(* PLC project Adressering.ecp, WAGO e!COCKPIT e!COCKPIT *)
(* stored: creationDateTime 2021-01-18T14:20:23.2110188, modificationDateTime 2021-01-18T11:51:27.6823754 *)

TYPE typVAV : STRUCT
  xReady : BOOL;  (* Status adr. *)
  xEnable : BOOL;  (* Enable MP blokk *)
  xAddress : BOOL;  (* Adresserer VAV *)
  xFailed : BOOL;  (* Tilbakemelding adressering (True = SerieNr inn og ut ikke stemmer) *)
  sSetStatus : STRING;  (* Status tilbakemelding naar adresseringen er i SET step *)
  sGetStatus : STRING;  (* Status tilbakemelding naar adresseringen er i GET step *)
  iSerialNr : typSerialNo;  (* Serie NR *)
  bPort : BYTE;  (* VAV Port *)
  bAddress : BYTE;  (* VAV Address *)
  rAirVolume_SP : REAL;  (* Settpunkt 0-100% *)
  rOutPosition : REAL;  (* Vinkel *)
  rOutAirVolume_perc : REAL;  (* Luftmengde i prosent *)
  rOutAirVolume_m3h : REAL;  (* Luftmengde i m3h *)
  wSensorValue : WORD;
  rVmin : REAL;
  rVmax : REAL;  (* Max vinkel *)
  xControlRangeIncreased : BOOL;
  xMecanicalOverload : BOOL;
  xActuatorHunting : BOOL;
  xSensorError : BOOL;
  xManualOpen : BOOL;
  xManualClose : BOOL;
  vMin : REAL;  (* Min luftmengde SP / 0-100 *)
  vNorm : REAL;  (* Settpunkt ved bevegelse / 0-100 *)
  vMax : REAL;  (* Maks luftmengde SP / 0-100 *)
  vSize : REAL;  (* Max kubikk *)
  vSetpoint_m3h : REAL;  (* SP% *)
  xdontoptimize : BOOL;  (* Fjerner VAV fra Optimizer *)
END_STRUCT;
END_TYPE

{attribute 'qualified_only'}
VAR_GLOBAL  (* STLV59_360 *)
  STLV59_A_360_001_OU001_SQ401_Max : REAL;  (* Max spjeldvinkel tilluft *)
  STLV59_A_360_001_OU001_SQ501_Max : REAL;  (* max spjeldvinkel avtrekk *)
  STLV59_A_360_002_SQ401 : typVAV := (xEnable := TRUE, vMin := 125, vNorm := 250, vMax := 500, vSize := 1060, bPort := 1, bAddress := 1, iSerialNr := (wYearAndWeek := 0, wDayAndNumber := 0, bTypeID := 0, bTestStation := 0));  (* / *)
  STLV59_A_360_014_SQ401 : typVAV := (xEnable := TRUE, vMin := 75, vNorm := 0, vMax := 300, vSize := 434, bPort := 1, bAddress := 2, iSerialNr := (wYearAndWeek := 0, wDayAndNumber := 0, bTypeID := 0, bTestStation := 0));  (* / *)
  STLV59_A_360_014_SQ501 : typVAV := (xEnable := TRUE, vMin := 75, vNorm := 0, vMax := 300, vSize := 434, bPort := 1, bAddress := 3, iSerialNr := (wYearAndWeek := 0, wDayAndNumber := 0, bTypeID := 0, bTestStation := 0));  (* / *)
  STLV59_A_360_103_SQ401 : typVAV := (xEnable := TRUE, vMin := 375, vNorm := 0, vMax := 1500, vSize := 3619, bPort := 1, bAddress := 4, iSerialNr := (wYearAndWeek := 0, wDayAndNumber := 0, bTypeID := 0, bTestStation := 0));  (* / *)
  STLV59_A_360_103_SQ402 : typVAV := (xEnable := TRUE, vMin := 375, vNorm := 0, vMax := 1500, vSize := 3619, bPort := 1, bAddress := 5, iSerialNr := (wYearAndWeek := 0, wDayAndNumber := 0, bTypeID := 0, bTestStation := 0));  (* / *)
  STLV59_A_360_103_SQ501 : typVAV := (xEnable := TRUE, vMin := 375, vNorm := 0, vMax := 1500, vSize := 3619, bPort := 1, bAddress := 6, iSerialNr := (wYearAndWeek := 0, wDayAndNumber := 0, bTypeID := 0, bTestStation := 0));  (* / *)
  STLV59_A_360_103_SQ502 : typVAV := (xEnable := TRUE, vMin := 375, vNorm := 0, vMax := 1500, vSize := 3619, bPort := 1, bAddress := 7, iSerialNr := (wYearAndWeek := 0, wDayAndNumber := 0, bTypeID := 0, bTestStation := 0));  (* / *)
  STLV59_A_360_002_SQ402 : typVAV := (xEnable := TRUE, vMin := 175, vNorm := 0, vMax := 700, vSize := 1060, bPort := 2, bAddress := 1, iSerialNr := (wYearAndWeek := 0, wDayAndNumber := 0, bTypeID := 0, bTestStation := 0));  (* / *)
  STLV59_A_360_002_SQ501 : typVAV := (xEnable := TRUE, vMin := 125, vNorm := 250, vMax := 500, vSize := 1060, bPort := 2, bAddress := 2, iSerialNr := (wYearAndWeek := 0, wDayAndNumber := 0, bTypeID := 0, bTestStation := 0));  (* / *)
  STLV59_A_360_002_SQ502 : typVAV := (xEnable := TRUE, vMin := 175, vNorm := 0, vMax := 700, vSize := 1060, bPort := 2, bAddress := 3, iSerialNr := (wYearAndWeek := 0, wDayAndNumber := 0, bTypeID := 0, bTestStation := 0));  (* / *)
  STLV59_A_360_006_SQ401 : typVAV := (xEnable := TRUE, vMin := 188, vNorm := 0, vMax := 750, vSize := 1060, bPort := 2, bAddress := 4, iSerialNr := (wYearAndWeek := 0, wDayAndNumber := 0, bTypeID := 0, bTestStation := 0));  (* / *)
  STLV59_A_360_008_SQ501 : typVAV := (xEnable := TRUE, vMin := 188, vNorm := 0, vMax := 750, vSize := 1060, bPort := 2, bAddress := 5, iSerialNr := (wYearAndWeek := 0, wDayAndNumber := 0, bTypeID := 0, bTestStation := 0));  (* / *)
  STLV59_A_360_011_SQ401 : typVAV := (xEnable := TRUE, vMin := 50, vNorm := 0, vMax := 200, vSize := 700, bPort := 2, bAddress := 6, iSerialNr := (wYearAndWeek := 0, wDayAndNumber := 0, bTypeID := 0, bTestStation := 0));  (* / *)
  STLV59_A_360_011_SQ501 : typVAV := (xEnable := TRUE, vMin := 50, vNorm := 0, vMax := 200, vSize := 265, bPort := 2, bAddress := 7, iSerialNr := (wYearAndWeek := 0, wDayAndNumber := 0, bTypeID := 0, bTestStation := 0));  (* / *)
  STLV59_A_360_T1U_SQ401 : typVAV := (xEnable := TRUE, vMin := 50, vNorm := 0, vMax := 200, vSize := 434, bPort := 2, bAddress := 8, iSerialNr := (wYearAndWeek := 0, wDayAndNumber := 0, bTypeID := 0, bTestStation := 0));  (* / *)
  STLV59_A_360_001_SQ401 : typVAV := (xEnable := TRUE, vMin := 25, vNorm := 100, vMax := 100, vSize := 265, bPort := 3, bAddress := 1, iSerialNr := (wYearAndWeek := 0, wDayAndNumber := 0, bTypeID := 0, bTestStation := 0));  (* / *)
  STLV59_A_360_001_SQ501 : typVAV := (xEnable := TRUE, vMin := 25, vNorm := 100, vMax := 100, vSize := 265, bPort := 3, bAddress := 2, iSerialNr := (wYearAndWeek := 0, wDayAndNumber := 0, bTypeID := 0, bTestStation := 0));  (* / *)
  STLV59_A_360_109_SQ401 : typVAV := (xEnable := TRUE, vMin := 200, vNorm := 200, vMax := 200, vSize := 434, bPort := 3, bAddress := 3, iSerialNr := (wYearAndWeek := 0, wDayAndNumber := 0, bTypeID := 0, bTestStation := 0));  (* / *)
  STLV59_A_360_110_SQ501 : typVAV := (xEnable := TRUE, vMin := 200, vNorm := 200, vMax := 200, vSize := 265, bPort := 3, bAddress := 4, iSerialNr := (wYearAndWeek := 0, wDayAndNumber := 0, bTypeID := 0, bTestStation := 0));  (* / *)
  STLV59_A_360_212_SQ401 : typVAV := (xEnable := TRUE, vMin := 63, vNorm := 0, vMax := 250, vSize := 700, bPort := 3, bAddress := 5, iSerialNr := (wYearAndWeek := 0, wDayAndNumber := 0, bTypeID := 0, bTestStation := 0));  (* / *)
  STLV59_A_360_212_SQ501 : typVAV := (xEnable := TRUE, vMin := 63, vNorm := 0, vMax := 250, vSize := 700, bPort := 3, bAddress := 6, iSerialNr := (wYearAndWeek := 0, wDayAndNumber := 0, bTypeID := 0, bTestStation := 0));  (* / *)
  STLV59_A_360_213_SQ401 : typVAV := (xEnable := TRUE, vMin := 138, vNorm := 0, vMax := 550, vSize := 70, bPort := 3, bAddress := 7, iSerialNr := (wYearAndWeek := 0, wDayAndNumber := 0, bTypeID := 0, bTestStation := 0));  (* / *)
  STLV59_A_360_213_SQ501 : typVAV := (xEnable := TRUE, vMin := 138, vNorm := 0, vMax := 550, vSize := 265, bPort := 3, bAddress := 8, iSerialNr := (wYearAndWeek := 0, wDayAndNumber := 0, bTypeID := 0, bTestStation := 0));  (* / *)
END_VAR

FUNCTION_BLOCK fbAutAd
  VAR_INPUT
    iSerialNr : typSerialNo;
    bPort : BYTE;
    bAddress : BYTE;
    xReset : BOOL;
    xNext : BOOL;
  END_VAR
  VAR_OUTPUT
    i : INT := 0;
    xFailed : BOOL;
    sSetStatus : STRING;
    sGetStatus : STRING;
  END_VAR
  VAR
    xLearn : BOOL;
    xRetry : BOOL;
    VAV_Addressing : fbMpBusAddressing;
  END_VAR

	//Resetter forgje VAVs verdier
	IF xReset THEN
		i:= 0;
		xRetry:= FALSE;
		xFailed:= FALSE;
		sSetStatus:= '';
		sGetStatus:= '';

//Begynner paa neste VAV
	ELSIF i<1 AND xNext THEN
		VAV_Addressing
		(
			bPortMpBus:= bPort,
			bAddress:= bAddress,
			typINSerialNo:= iSerialNr,
			xLearn:= xLearn
		);
		i:= 1;

//Skriver rett port og adresse til VAV naar blokken er klar
	ELSIF VAV_Addressing.xReady AND i=1 THEN
		VAV_Addressing
		(
			xSet:= TRUE,
			xLearn:= xLearn
		);
		i:= 2;

//Spoer etter serie nr som hoerer til port og adresse
	ELSIF VAV_Addressing.xReady AND i=2 THEN
		sSetStatus:= VAV_Addressing.sStatus;
		VAV_Addressing
		(
			xGetSerialNO:= TRUE,
			xLearn:= xLearn
		);
		i:= 3;

//Sjekker om serie nr. som tilhoerer port og adressen stemmer
	ELSIF VAV_Addressing.xReady AND i=3 THEN
		sGetStatus:= VAV_Addressing.sStatus;
		//Sjekker om serie nr stemmer
		IF xRetry AND VAV_Addressing.typOUTSerialNo.wYearAndWeek <> iSerialNr.wYearAndWeek OR VAV_Addressing.typOUTSerialNo.wDayAndNumber <> iSerialNr.wDayAndNumber OR VAV_Addressing.typOUTSerialNo.bTypeID <> iSerialNr.bTypeID OR VAV_Addressing.typOUTSerialNo.bTestStation <> iSerialNr.bTestStation THEN
			xRetry:= FALSE;
			xFailed:= TRUE;
			i:=4;
		ELSIF VAV_Addressing.typOUTSerialNo.wYearAndWeek <> iSerialNr.wYearAndWeek OR VAV_Addressing.typOUTSerialNo.wDayAndNumber <> iSerialNr.wDayAndNumber OR VAV_Addressing.typOUTSerialNo.bTypeID <> iSerialNr.bTypeID OR VAV_Addressing.typOUTSerialNo.bTestStation <> iSerialNr.bTestStation THEN
			xRetry:= TRUE;
			i:=1;
		ELSE
			i:=4;
		END_IF

//Resetter xSet og xGet, og Setter Port, adresse og serie nr. og henter status
	ELSE
		VAV_Addressing
		(
			bPortMpBus:= bPort,
			bAddress:= bAddress,
			typINSerialNo:= iSerialNr,
			xLearn:= xLearn,
			xSet:= FALSE,
			xGetSerialNO:= FALSE,
			xLearn:= xLearn
		);
	END_IF
				
END_FUNCTION_BLOCK

PROGRAM PRG_360_VAV_Adressering
  VAR
    xReset : BOOL;
    xRun : BOOL;
    xInit : BOOL := TRUE;
    Auto : fbAutAd;
    iLinje : INT;  (* Linje som skal adresseres *)
    iVAV : INT := 1;  (* VAV(adr.) som adresseres *)
  END_VAR

					IF xReset THEN
	Auto(xReset:= TRUE);
	xInit:= TRUE;
	xReset:= FALSE;
ELSIF xRun THEN

	IF STLV59_360.STLV59_A_360_002_SQ401.xAddress OR (iLinje = 1 AND iVAV = 1) THEN

		IF xInit THEN
			STLV59_360.STLV59_A_360_002_SQ401.xEnable:= FALSE;
			Auto(
				bPort:= STLV59_360.STLV59_A_360_002_SQ401.bPort,
				bAddress:= STLV59_360.STLV59_A_360_002_SQ401.bAddress,
				iSerialNr:= STLV59_360.STLV59_A_360_002_SQ401.iSerialNr,
				xNext:= TRUE,
				xReset:= FALSE
				);
			xInit:= FALSE;

		ELSIF Auto.i=4 THEN
			STLV59_360.STLV59_A_360_002_SQ401.sSetStatus:= Auto.sSetStatus;
				STLV59_360.STLV59_A_360_002_SQ401.sGetStatus:= Auto.sGetStatus;
				STLV59_360.STLV59_A_360_002_SQ401.xFailed:= Auto.xFailed;
				STLV59_360.STLV59_A_360_002_SQ401.xAddress:= FALSE;
				STLV59_360.STLV59_A_360_002_SQ401.xEnable:= TRUE;
				xReset:= TRUE;
				iVAV:=iVAV+1;

			ELSE
				Auto(xNext:= FALSE);
			END_IF

	ELSIF STLV59_360.STLV59_A_360_014_SQ401.xAddress OR (iLinje = 1 AND iVAV = 2) THEN

		IF xInit THEN
			STLV59_360.STLV59_A_360_014_SQ401.xEnable:= FALSE;
			Auto(
				bPort:= STLV59_360.STLV59_A_360_014_SQ401.bPort,
				bAddress:= STLV59_360.STLV59_A_360_014_SQ401.bAddress,
				iSerialNr:= STLV59_360.STLV59_A_360_014_SQ401.iSerialNr,
				xNext:= TRUE,
				xReset:= FALSE
				);
			xInit:= FALSE;

		ELSIF Auto.i=4 THEN
			STLV59_360.STLV59_A_360_014_SQ401.sSetStatus:= Auto.sSetStatus;
				STLV59_360.STLV59_A_360_014_SQ401.sGetStatus:= Auto.sGetStatus;
				STLV59_360.STLV59_A_360_014_SQ401.xFailed:= Auto.xFailed;
				STLV59_360.STLV59_A_360_014_SQ401.xAddress:= FALSE;
				STLV59_360.STLV59_A_360_014_SQ401.xEnable:= TRUE;
				xReset:= TRUE;
				iVAV:=iVAV+1;

			ELSE
				Auto(xNext:= FALSE);
			END_IF

	ELSIF STLV59_360.STLV59_A_360_014_SQ501.xAddress OR (iLinje = 1 AND iVAV = 3) THEN

		IF xInit THEN
			STLV59_360.STLV59_A_360_014_SQ501.xEnable:= FALSE;
			Auto(
				bPort:= STLV59_360.STLV59_A_360_014_SQ501.bPort,
				bAddress:= STLV59_360.STLV59_A_360_014_SQ501.bAddress,
				iSerialNr:= STLV59_360.STLV59_A_360_014_SQ501.iSerialNr,
				xNext:= TRUE,
				xReset:= FALSE
				);
			xInit:= FALSE;

		ELSIF Auto.i=4 THEN
			STLV59_360.STLV59_A_360_014_SQ501.sSetStatus:= Auto.sSetStatus;
				STLV59_360.STLV59_A_360_014_SQ501.sGetStatus:= Auto.sGetStatus;
				STLV59_360.STLV59_A_360_014_SQ501.xFailed:= Auto.xFailed;
				STLV59_360.STLV59_A_360_014_SQ501.xAddress:= FALSE;
				STLV59_360.STLV59_A_360_014_SQ501.xEnable:= TRUE;
				xReset:= TRUE;
				iVAV:=iVAV+1;

			ELSE
				Auto(xNext:= FALSE);
			END_IF

	ELSIF STLV59_360.STLV59_A_360_103_SQ401.xAddress OR (iLinje = 1 AND iVAV = 4) THEN

		IF xInit THEN
			STLV59_360.STLV59_A_360_103_SQ401.xEnable:= FALSE;
			Auto(
				bPort:= STLV59_360.STLV59_A_360_103_SQ401.bPort,
				bAddress:= STLV59_360.STLV59_A_360_103_SQ401.bAddress,
				iSerialNr:= STLV59_360.STLV59_A_360_103_SQ401.iSerialNr,
				xNext:= TRUE,
				xReset:= FALSE
				);
			xInit:= FALSE;

		ELSIF Auto.i=4 THEN
			STLV59_360.STLV59_A_360_103_SQ401.sSetStatus:= Auto.sSetStatus;
				STLV59_360.STLV59_A_360_103_SQ401.sGetStatus:= Auto.sGetStatus;
				STLV59_360.STLV59_A_360_103_SQ401.xFailed:= Auto.xFailed;
				STLV59_360.STLV59_A_360_103_SQ401.xAddress:= FALSE;
				STLV59_360.STLV59_A_360_103_SQ401.xEnable:= TRUE;
				xReset:= TRUE;
				iVAV:=iVAV+1;

			ELSE
				Auto(xNext:= FALSE);
			END_IF

	ELSIF STLV59_360.STLV59_A_360_103_SQ402.xAddress OR (iLinje = 1 AND iVAV = 5) THEN

		IF xInit THEN
			STLV59_360.STLV59_A_360_103_SQ402.xEnable:= FALSE;
			Auto(
				bPort:= STLV59_360.STLV59_A_360_103_SQ402.bPort,
				bAddress:= STLV59_360.STLV59_A_360_103_SQ402.bAddress,
				iSerialNr:= STLV59_360.STLV59_A_360_103_SQ402.iSerialNr,
				xNext:= TRUE,
				xReset:= FALSE
				);
			xInit:= FALSE;

		ELSIF Auto.i=4 THEN
			STLV59_360.STLV59_A_360_103_SQ402.sSetStatus:= Auto.sSetStatus;
				STLV59_360.STLV59_A_360_103_SQ402.sGetStatus:= Auto.sGetStatus;
				STLV59_360.STLV59_A_360_103_SQ402.xFailed:= Auto.xFailed;
				STLV59_360.STLV59_A_360_103_SQ402.xAddress:= FALSE;
				STLV59_360.STLV59_A_360_103_SQ402.xEnable:= TRUE;
				xReset:= TRUE;
				iVAV:=iVAV+1;

			ELSE
				Auto(xNext:= FALSE);
			END_IF

	ELSIF STLV59_360.STLV59_A_360_103_SQ501.xAddress OR (iLinje = 1 AND iVAV = 6) THEN

		IF xInit THEN
			STLV59_360.STLV59_A_360_103_SQ501.xEnable:= FALSE;
			Auto(
				bPort:= STLV59_360.STLV59_A_360_103_SQ501.bPort,
				bAddress:= STLV59_360.STLV59_A_360_103_SQ501.bAddress,
				iSerialNr:= STLV59_360.STLV59_A_360_103_SQ501.iSerialNr,
				xNext:= TRUE,
				xReset:= FALSE
				);
			xInit:= FALSE;

		ELSIF Auto.i=4 THEN
			STLV59_360.STLV59_A_360_103_SQ501.sSetStatus:= Auto.sSetStatus;
				STLV59_360.STLV59_A_360_103_SQ501.sGetStatus:= Auto.sGetStatus;
				STLV59_360.STLV59_A_360_103_SQ501.xFailed:= Auto.xFailed;
				STLV59_360.STLV59_A_360_103_SQ501.xAddress:= FALSE;
				STLV59_360.STLV59_A_360_103_SQ501.xEnable:= TRUE;
				xReset:= TRUE;
				iVAV:=iVAV+1;

			ELSE
				Auto(xNext:= FALSE);
			END_IF

	ELSIF STLV59_360.STLV59_A_360_103_SQ502.xAddress OR (iLinje = 1 AND iVAV = 7) THEN

		IF xInit THEN
			STLV59_360.STLV59_A_360_103_SQ502.xEnable:= FALSE;
			Auto(
				bPort:= STLV59_360.STLV59_A_360_103_SQ502.bPort,
				bAddress:= STLV59_360.STLV59_A_360_103_SQ502.bAddress,
				iSerialNr:= STLV59_360.STLV59_A_360_103_SQ502.iSerialNr,
				xNext:= TRUE,
				xReset:= FALSE
				);
			xInit:= FALSE;

		ELSIF Auto.i=4 THEN
			STLV59_360.STLV59_A_360_103_SQ502.sSetStatus:= Auto.sSetStatus;
				STLV59_360.STLV59_A_360_103_SQ502.sGetStatus:= Auto.sGetStatus;
				STLV59_360.STLV59_A_360_103_SQ502.xFailed:= Auto.xFailed;
				STLV59_360.STLV59_A_360_103_SQ502.xAddress:= FALSE;
				STLV59_360.STLV59_A_360_103_SQ502.xEnable:= TRUE;
				xReset:= TRUE;
				iVAV:=iVAV+1;

			ELSE
				Auto(xNext:= FALSE);
			END_IF

	ELSIF STLV59_360.STLV59_A_360_002_SQ402.xAddress OR (iLinje = 2 AND iVAV = 1) THEN

		IF xInit THEN
			STLV59_360.STLV59_A_360_002_SQ402.xEnable:= FALSE;
			Auto(
				bPort:= STLV59_360.STLV59_A_360_002_SQ402.bPort,
				bAddress:= STLV59_360.STLV59_A_360_002_SQ402.bAddress,
				iSerialNr:= STLV59_360.STLV59_A_360_002_SQ402.iSerialNr,
				xNext:= TRUE,
				xReset:= FALSE
				);
			xInit:= FALSE;

		ELSIF Auto.i=4 THEN
			STLV59_360.STLV59_A_360_002_SQ402.sSetStatus:= Auto.sSetStatus;
				STLV59_360.STLV59_A_360_002_SQ402.sGetStatus:= Auto.sGetStatus;
				STLV59_360.STLV59_A_360_002_SQ402.xFailed:= Auto.xFailed;
				STLV59_360.STLV59_A_360_002_SQ402.xAddress:= FALSE;
				STLV59_360.STLV59_A_360_002_SQ402.xEnable:= TRUE;
				xReset:= TRUE;
				iVAV:=iVAV+1;

			ELSE
				Auto(xNext:= FALSE);
			END_IF

	ELSIF STLV59_360.STLV59_A_360_002_SQ501.xAddress OR (iLinje = 2 AND iVAV = 2) THEN

		IF xInit THEN
			STLV59_360.STLV59_A_360_002_SQ501.xEnable:= FALSE;
			Auto(
				bPort:= STLV59_360.STLV59_A_360_002_SQ501.bPort,
				bAddress:= STLV59_360.STLV59_A_360_002_SQ501.bAddress,
				iSerialNr:= STLV59_360.STLV59_A_360_002_SQ501.iSerialNr,
				xNext:= TRUE,
				xReset:= FALSE
				);
			xInit:= FALSE;

		ELSIF Auto.i=4 THEN
			STLV59_360.STLV59_A_360_002_SQ501.sSetStatus:= Auto.sSetStatus;
				STLV59_360.STLV59_A_360_002_SQ501.sGetStatus:= Auto.sGetStatus;
				STLV59_360.STLV59_A_360_002_SQ501.xFailed:= Auto.xFailed;
				STLV59_360.STLV59_A_360_002_SQ501.xAddress:= FALSE;
				STLV59_360.STLV59_A_360_002_SQ501.xEnable:= TRUE;
				xReset:= TRUE;
				iVAV:=iVAV+1;

			ELSE
				Auto(xNext:= FALSE);
			END_IF

	ELSIF STLV59_360.STLV59_A_360_002_SQ502.xAddress OR (iLinje = 2 AND iVAV = 3) THEN

		IF xInit THEN
			STLV59_360.STLV59_A_360_002_SQ502.xEnable:= FALSE;
			Auto(
				bPort:= STLV59_360.STLV59_A_360_002_SQ502.bPort,
				bAddress:= STLV59_360.STLV59_A_360_002_SQ502.bAddress,
				iSerialNr:= STLV59_360.STLV59_A_360_002_SQ502.iSerialNr,
				xNext:= TRUE,
				xReset:= FALSE
				);
			xInit:= FALSE;

		ELSIF Auto.i=4 THEN
			STLV59_360.STLV59_A_360_002_SQ502.sSetStatus:= Auto.sSetStatus;
				STLV59_360.STLV59_A_360_002_SQ502.sGetStatus:= Auto.sGetStatus;
				STLV59_360.STLV59_A_360_002_SQ502.xFailed:= Auto.xFailed;
				STLV59_360.STLV59_A_360_002_SQ502.xAddress:= FALSE;
				STLV59_360.STLV59_A_360_002_SQ502.xEnable:= TRUE;
				xReset:= TRUE;
				iVAV:=iVAV+1;

			ELSE
				Auto(xNext:= FALSE);
			END_IF

	ELSIF STLV59_360.STLV59_A_360_006_SQ401.xAddress OR (iLinje = 2 AND iVAV = 4) THEN

		IF xInit THEN
			STLV59_360.STLV59_A_360_006_SQ401.xEnable:= FALSE;
			Auto(
				bPort:= STLV59_360.STLV59_A_360_006_SQ401.bPort,
				bAddress:= STLV59_360.STLV59_A_360_006_SQ401.bAddress,
				iSerialNr:= STLV59_360.STLV59_A_360_006_SQ401.iSerialNr,
				xNext:= TRUE,
				xReset:= FALSE
				);
			xInit:= FALSE;

		ELSIF Auto.i=4 THEN
			STLV59_360.STLV59_A_360_006_SQ401.sSetStatus:= Auto.sSetStatus;
				STLV59_360.STLV59_A_360_006_SQ401.sGetStatus:= Auto.sGetStatus;
				STLV59_360.STLV59_A_360_006_SQ401.xFailed:= Auto.xFailed;
				STLV59_360.STLV59_A_360_006_SQ401.xAddress:= FALSE;
				STLV59_360.STLV59_A_360_006_SQ401.xEnable:= TRUE;
				xReset:= TRUE;
				iVAV:=iVAV+1;

			ELSE
				Auto(xNext:= FALSE);
			END_IF

	ELSIF STLV59_360.STLV59_A_360_008_SQ501.xAddress OR (iLinje = 2 AND iVAV = 5) THEN

		IF xInit THEN
			STLV59_360.STLV59_A_360_008_SQ501.xEnable:= FALSE;
			Auto(
				bPort:= STLV59_360.STLV59_A_360_008_SQ501.bPort,
				bAddress:= STLV59_360.STLV59_A_360_008_SQ501.bAddress,
				iSerialNr:= STLV59_360.STLV59_A_360_008_SQ501.iSerialNr,
				xNext:= TRUE,
				xReset:= FALSE
				);
			xInit:= FALSE;

		ELSIF Auto.i=4 THEN
			STLV59_360.STLV59_A_360_008_SQ501.sSetStatus:= Auto.sSetStatus;
				STLV59_360.STLV59_A_360_008_SQ501.sGetStatus:= Auto.sGetStatus;
				STLV59_360.STLV59_A_360_008_SQ501.xFailed:= Auto.xFailed;
				STLV59_360.STLV59_A_360_008_SQ501.xAddress:= FALSE;
				STLV59_360.STLV59_A_360_008_SQ501.xEnable:= TRUE;
				xReset:= TRUE;
				iVAV:=iVAV+1;

			ELSE
				Auto(xNext:= FALSE);
			END_IF

	ELSIF STLV59_360.STLV59_A_360_011_SQ401.xAddress OR (iLinje = 2 AND iVAV = 6) THEN

		IF xInit THEN
			STLV59_360.STLV59_A_360_011_SQ401.xEnable:= FALSE;
			Auto(
				bPort:= STLV59_360.STLV59_A_360_011_SQ401.bPort,
				bAddress:= STLV59_360.STLV59_A_360_011_SQ401.bAddress,
				iSerialNr:= STLV59_360.STLV59_A_360_011_SQ401.iSerialNr,
				xNext:= TRUE,
				xReset:= FALSE
				);
			xInit:= FALSE;

		ELSIF Auto.i=4 THEN
			STLV59_360.STLV59_A_360_011_SQ401.sSetStatus:= Auto.sSetStatus;
				STLV59_360.STLV59_A_360_011_SQ401.sGetStatus:= Auto.sGetStatus;
				STLV59_360.STLV59_A_360_011_SQ401.xFailed:= Auto.xFailed;
				STLV59_360.STLV59_A_360_011_SQ401.xAddress:= FALSE;
				STLV59_360.STLV59_A_360_011_SQ401.xEnable:= TRUE;
				xReset:= TRUE;
				iVAV:=iVAV+1;

			ELSE
				Auto(xNext:= FALSE);
			END_IF

	ELSIF STLV59_360.STLV59_A_360_011_SQ501.xAddress OR (iLinje = 2 AND iVAV = 7) THEN

		IF xInit THEN
			STLV59_360.STLV59_A_360_011_SQ501.xEnable:= FALSE;
			Auto(
				bPort:= STLV59_360.STLV59_A_360_011_SQ501.bPort,
				bAddress:= STLV59_360.STLV59_A_360_011_SQ501.bAddress,
				iSerialNr:= STLV59_360.STLV59_A_360_011_SQ501.iSerialNr,
				xNext:= TRUE,
				xReset:= FALSE
				);
			xInit:= FALSE;

		ELSIF Auto.i=4 THEN
			STLV59_360.STLV59_A_360_011_SQ501.sSetStatus:= Auto.sSetStatus;
				STLV59_360.STLV59_A_360_011_SQ501.sGetStatus:= Auto.sGetStatus;
				STLV59_360.STLV59_A_360_011_SQ501.xFailed:= Auto.xFailed;
				STLV59_360.STLV59_A_360_011_SQ501.xAddress:= FALSE;
				STLV59_360.STLV59_A_360_011_SQ501.xEnable:= TRUE;
				xReset:= TRUE;
				iVAV:=iVAV+1;

			ELSE
				Auto(xNext:= FALSE);
			END_IF

	ELSIF STLV59_360.STLV59_A_360_T1U_SQ401.xAddress OR (iLinje = 2 AND iVAV = 8) THEN

		IF xInit THEN
			STLV59_360.STLV59_A_360_T1U_SQ401.xEnable:= FALSE;
			Auto(
				bPort:= STLV59_360.STLV59_A_360_T1U_SQ401.bPort,
				bAddress:= STLV59_360.STLV59_A_360_T1U_SQ401.bAddress,
				iSerialNr:= STLV59_360.STLV59_A_360_T1U_SQ401.iSerialNr,
				xNext:= TRUE,
				xReset:= FALSE
				);
			xInit:= FALSE;

		ELSIF Auto.i=4 THEN
			STLV59_360.STLV59_A_360_T1U_SQ401.sSetStatus:= Auto.sSetStatus;
				STLV59_360.STLV59_A_360_T1U_SQ401.sGetStatus:= Auto.sGetStatus;
				STLV59_360.STLV59_A_360_T1U_SQ401.xFailed:= Auto.xFailed;
				STLV59_360.STLV59_A_360_T1U_SQ401.xAddress:= FALSE;
				STLV59_360.STLV59_A_360_T1U_SQ401.xEnable:= TRUE;
				xReset:= TRUE;
				iVAV:=iVAV+1;

			ELSE
				Auto(xNext:= FALSE);
			END_IF

	ELSIF STLV59_360.STLV59_A_360_001_SQ401.xAddress OR (iLinje = 3 AND iVAV = 1) THEN

		IF xInit THEN
			STLV59_360.STLV59_A_360_001_SQ401.xEnable:= FALSE;
			Auto(
				bPort:= STLV59_360.STLV59_A_360_001_SQ401.bPort,
				bAddress:= STLV59_360.STLV59_A_360_001_SQ401.bAddress,
				iSerialNr:= STLV59_360.STLV59_A_360_001_SQ401.iSerialNr,
				xNext:= TRUE,
				xReset:= FALSE
				);
			xInit:= FALSE;

		ELSIF Auto.i=4 THEN
			STLV59_360.STLV59_A_360_001_SQ401.sSetStatus:= Auto.sSetStatus;
				STLV59_360.STLV59_A_360_001_SQ401.sGetStatus:= Auto.sGetStatus;
				STLV59_360.STLV59_A_360_001_SQ401.xFailed:= Auto.xFailed;
				STLV59_360.STLV59_A_360_001_SQ401.xAddress:= FALSE;
				STLV59_360.STLV59_A_360_001_SQ401.xEnable:= TRUE;
				xReset:= TRUE;
				iVAV:=iVAV+1;

			ELSE
				Auto(xNext:= FALSE);
			END_IF

	ELSIF STLV59_360.STLV59_A_360_001_SQ501.xAddress OR (iLinje = 3 AND iVAV = 2) THEN

		IF xInit THEN
			STLV59_360.STLV59_A_360_001_SQ501.xEnable:= FALSE;
			Auto(
				bPort:= STLV59_360.STLV59_A_360_001_SQ501.bPort,
				bAddress:= STLV59_360.STLV59_A_360_001_SQ501.bAddress,
				iSerialNr:= STLV59_360.STLV59_A_360_001_SQ501.iSerialNr,
				xNext:= TRUE,
				xReset:= FALSE
				);
			xInit:= FALSE;

		ELSIF Auto.i=4 THEN
			STLV59_360.STLV59_A_360_001_SQ501.sSetStatus:= Auto.sSetStatus;
				STLV59_360.STLV59_A_360_001_SQ501.sGetStatus:= Auto.sGetStatus;
				STLV59_360.STLV59_A_360_001_SQ501.xFailed:= Auto.xFailed;
				STLV59_360.STLV59_A_360_001_SQ501.xAddress:= FALSE;
				STLV59_360.STLV59_A_360_001_SQ501.xEnable:= TRUE;
				xReset:= TRUE;
				iVAV:=iVAV+1;

			ELSE
				Auto(xNext:= FALSE);
			END_IF

	ELSIF STLV59_360.STLV59_A_360_109_SQ401.xAddress OR (iLinje = 3 AND iVAV = 3) THEN

		IF xInit THEN
			STLV59_360.STLV59_A_360_109_SQ401.xEnable:= FALSE;
			Auto(
				bPort:= STLV59_360.STLV59_A_360_109_SQ401.bPort,
				bAddress:= STLV59_360.STLV59_A_360_109_SQ401.bAddress,
				iSerialNr:= STLV59_360.STLV59_A_360_109_SQ401.iSerialNr,
				xNext:= TRUE,
				xReset:= FALSE
				);
			xInit:= FALSE;

		ELSIF Auto.i=4 THEN
			STLV59_360.STLV59_A_360_109_SQ401.sSetStatus:= Auto.sSetStatus;
				STLV59_360.STLV59_A_360_109_SQ401.sGetStatus:= Auto.sGetStatus;
				STLV59_360.STLV59_A_360_109_SQ401.xFailed:= Auto.xFailed;
				STLV59_360.STLV59_A_360_109_SQ401.xAddress:= FALSE;
				STLV59_360.STLV59_A_360_109_SQ401.xEnable:= TRUE;
				xReset:= TRUE;
				iVAV:=iVAV+1;

			ELSE
				Auto(xNext:= FALSE);
			END_IF

	ELSIF STLV59_360.STLV59_A_360_110_SQ501.xAddress OR (iLinje = 3 AND iVAV = 4) THEN

		IF xInit THEN
			STLV59_360.STLV59_A_360_110_SQ501.xEnable:= FALSE;
			Auto(
				bPort:= STLV59_360.STLV59_A_360_110_SQ501.bPort,
				bAddress:= STLV59_360.STLV59_A_360_110_SQ501.bAddress,
				iSerialNr:= STLV59_360.STLV59_A_360_110_SQ501.iSerialNr,
				xNext:= TRUE,
				xReset:= FALSE
				);
			xInit:= FALSE;

		ELSIF Auto.i=4 THEN
			STLV59_360.STLV59_A_360_110_SQ501.sSetStatus:= Auto.sSetStatus;
				STLV59_360.STLV59_A_360_110_SQ501.sGetStatus:= Auto.sGetStatus;
				STLV59_360.STLV59_A_360_110_SQ501.xFailed:= Auto.xFailed;
				STLV59_360.STLV59_A_360_110_SQ501.xAddress:= FALSE;
				STLV59_360.STLV59_A_360_110_SQ501.xEnable:= TRUE;
				xReset:= TRUE;
				iVAV:=iVAV+1;

			ELSE
				Auto(xNext:= FALSE);
			END_IF

	ELSIF STLV59_360.STLV59_A_360_212_SQ401.xAddress OR (iLinje = 3 AND iVAV = 5) THEN

		IF xInit THEN
			STLV59_360.STLV59_A_360_212_SQ401.xEnable:= FALSE;
			Auto(
				bPort:= STLV59_360.STLV59_A_360_212_SQ401.bPort,
				bAddress:= STLV59_360.STLV59_A_360_212_SQ401.bAddress,
				iSerialNr:= STLV59_360.STLV59_A_360_212_SQ401.iSerialNr,
				xNext:= TRUE,
				xReset:= FALSE
				);
			xInit:= FALSE;

		ELSIF Auto.i=4 THEN
			STLV59_360.STLV59_A_360_212_SQ401.sSetStatus:= Auto.sSetStatus;
				STLV59_360.STLV59_A_360_212_SQ401.sGetStatus:= Auto.sGetStatus;
				STLV59_360.STLV59_A_360_212_SQ401.xFailed:= Auto.xFailed;
				STLV59_360.STLV59_A_360_212_SQ401.xAddress:= FALSE;
				STLV59_360.STLV59_A_360_212_SQ401.xEnable:= TRUE;
				xReset:= TRUE;
				iVAV:=iVAV+1;

			ELSE
				Auto(xNext:= FALSE);
			END_IF

	ELSIF STLV59_360.STLV59_A_360_212_SQ501.xAddress OR (iLinje = 3 AND iVAV = 6) THEN

		IF xInit THEN
			STLV59_360.STLV59_A_360_212_SQ501.xEnable:= FALSE;
			Auto(
				bPort:= STLV59_360.STLV59_A_360_212_SQ501.bPort,
				bAddress:= STLV59_360.STLV59_A_360_212_SQ501.bAddress,
				iSerialNr:= STLV59_360.STLV59_A_360_212_SQ501.iSerialNr,
				xNext:= TRUE,
				xReset:= FALSE
				);
			xInit:= FALSE;

		ELSIF Auto.i=4 THEN
			STLV59_360.STLV59_A_360_212_SQ501.sSetStatus:= Auto.sSetStatus;
				STLV59_360.STLV59_A_360_212_SQ501.sGetStatus:= Auto.sGetStatus;
				STLV59_360.STLV59_A_360_212_SQ501.xFailed:= Auto.xFailed;
				STLV59_360.STLV59_A_360_212_SQ501.xAddress:= FALSE;
				STLV59_360.STLV59_A_360_212_SQ501.xEnable:= TRUE;
				xReset:= TRUE;
				iVAV:=iVAV+1;

			ELSE
				Auto(xNext:= FALSE);
			END_IF

	ELSIF STLV59_360.STLV59_A_360_213_SQ401.xAddress OR (iLinje = 3 AND iVAV = 7) THEN

		IF xInit THEN
			STLV59_360.STLV59_A_360_213_SQ401.xEnable:= FALSE;
			Auto(
				bPort:= STLV59_360.STLV59_A_360_213_SQ401.bPort,
				bAddress:= STLV59_360.STLV59_A_360_213_SQ401.bAddress,
				iSerialNr:= STLV59_360.STLV59_A_360_213_SQ401.iSerialNr,
				xNext:= TRUE,
				xReset:= FALSE
				);
			xInit:= FALSE;

		ELSIF Auto.i=4 THEN
			STLV59_360.STLV59_A_360_213_SQ401.sSetStatus:= Auto.sSetStatus;
				STLV59_360.STLV59_A_360_213_SQ401.sGetStatus:= Auto.sGetStatus;
				STLV59_360.STLV59_A_360_213_SQ401.xFailed:= Auto.xFailed;
				STLV59_360.STLV59_A_360_213_SQ401.xAddress:= FALSE;
				STLV59_360.STLV59_A_360_213_SQ401.xEnable:= TRUE;
				xReset:= TRUE;
				iVAV:=iVAV+1;

			ELSE
				Auto(xNext:= FALSE);
			END_IF

	ELSIF STLV59_360.STLV59_A_360_213_SQ501.xAddress OR (iLinje = 3 AND iVAV = 8) THEN

		IF xInit THEN
			STLV59_360.STLV59_A_360_213_SQ501.xEnable:= FALSE;
			Auto(
				bPort:= STLV59_360.STLV59_A_360_213_SQ501.bPort,
				bAddress:= STLV59_360.STLV59_A_360_213_SQ501.bAddress,
				iSerialNr:= STLV59_360.STLV59_A_360_213_SQ501.iSerialNr,
				xNext:= TRUE,
				xReset:= FALSE
				);
			xInit:= FALSE;

		ELSIF Auto.i=4 THEN
			STLV59_360.STLV59_A_360_213_SQ501.sSetStatus:= Auto.sSetStatus;
				STLV59_360.STLV59_A_360_213_SQ501.sGetStatus:= Auto.sGetStatus;
				STLV59_360.STLV59_A_360_213_SQ501.xFailed:= Auto.xFailed;
				STLV59_360.STLV59_A_360_213_SQ501.xAddress:= FALSE;
				STLV59_360.STLV59_A_360_213_SQ501.xEnable:= TRUE;
				xReset:= TRUE;
				iVAV:=iVAV+1;

			ELSE
				Auto(xNext:= FALSE);
			END_IF

	ELSIF iVAV > 8 THEN
			iVAV:= 0;
		ELSIF iVAV > 0  THEN
			iVAV:= (iVAV+1);
		END_IF
END_IF

				
END_PROGRAM

PROGRAM PRG_360_MP1
  VAR
    xSet : BOOL;  (* Felles *)
    xRead : BOOL;
    FbMpbusMaster_1 : FbMpbusMaster;  (* Master *)
    oStatus_M1 : WagoSysErrorBase.FbResult;
    sStatus_M1 : STRING;
    FbMpbus_1 : FbMpBusVav;  (* Linje 1. Adresse 1. VAV STLV59_A_360_002_SQ401 *)
    oStatus_1 : WagoSysErrorBase.FbResult;
    sStatus_1 : STRING;
    FbMpbus_2 : FbMpBusVav;  (* Linje 1. Adresse 2. VAV STLV59_A_360_014_SQ401 *)
    oStatus_2 : WagoSysErrorBase.FbResult;
    sStatus_2 : STRING;
    FbMpbus_3 : FbMpBusVav;  (* Linje 1. Adresse 3. VAV STLV59_A_360_014_SQ501 *)
    oStatus_3 : WagoSysErrorBase.FbResult;
    sStatus_3 : STRING;
    FbMpbus_4 : FbMpBusVav;  (* Linje 1. Adresse 4. VAV STLV59_A_360_103_SQ401 *)
    oStatus_4 : WagoSysErrorBase.FbResult;
    sStatus_4 : STRING;
    FbMpbus_5 : FbMpBusVav;  (* Linje 1. Adresse 5. VAV STLV59_A_360_103_SQ402 *)
    oStatus_5 : WagoSysErrorBase.FbResult;
    sStatus_5 : STRING;
    FbMpbus_6 : FbMpBusVav;  (* Linje 1. Adresse 6. VAV STLV59_A_360_103_SQ501 *)
    oStatus_6 : WagoSysErrorBase.FbResult;
    sStatus_6 : STRING;
    FbMpbus_7 : FbMpBusVav;  (* Linje 1. Adresse 7. VAV STLV59_A_360_103_SQ502 *)
    oStatus_7 : WagoSysErrorBase.FbResult;
    sStatus_7 : STRING;
  END_VAR

(* CFC diagram, written out as Structured Text *)
FbMpbusMaster_1(I_Port := IoConfig_Globals.MP_Bus_Master, bPortMpBus := 1);
oStatus_M1 := FbMpbusMaster_1.oStatus;
sStatus_M1 := FbMpbusMaster_1.sStatus;
(* STLV59_A_360_002_SQ401 *)
FbMpbus_1(xEnable := STLV59_360.STLV59_A_360_002_SQ401.xEnable, bPortMpBus := 1, bAddress := 1, tCycleTime := t#500ms, rAirVolume := STLV59_360.STLV59_A_360_002_SQ401.rAirVolume_SP, rMinAirVolume := 0, rMaxAirVolume := 100, xSet := xSet, xRead := xRead, bSensorType := 0, xManualOpen := STLV59_360.STLV59_A_360_002_SQ401.xManualOpen, xManualClose := STLV59_360.STLV59_A_360_002_SQ401.xManualClose);
oStatus_1 := FbMpbus_1.oStatus;
sStatus_1 := FbMpbus_1.sStatus;
STLV59_360.STLV59_A_360_002_SQ401.xReady := FbMpbus_1.xReady;
STLV59_360.STLV59_A_360_002_SQ401.rOutPosition := FbMpbus_1.rOutPosition;
STLV59_360.STLV59_A_360_002_SQ401.rOutAirVolume_perc := FbMpbus_1.rOutAirVolume_perc;
STLV59_360.STLV59_A_360_002_SQ401.rOutAirVolume_m3h := FbMpbus_1.rOutAirVolume_m3_h;
STLV59_360.STLV59_A_360_002_SQ401.wSensorValue := FbMpbus_1.wSensorValue;
STLV59_360.STLV59_A_360_002_SQ401.rVmin := FbMpbus_1.rVmin;
STLV59_360.STLV59_A_360_002_SQ401.rVmax := FbMpbus_1.rVmax;
STLV59_360.STLV59_A_360_002_SQ401.xControlRangeIncreased := FbMpbus_1.xControlRangeIncreased;
STLV59_360.STLV59_A_360_002_SQ401.xMecanicalOverload := FbMpbus_1.xMecanicalOverload;
STLV59_360.STLV59_A_360_002_SQ401.xActuatorHunting := FbMpbus_1.xActuatorHunting;
STLV59_360.STLV59_A_360_002_SQ401.xSensorError := FbMpbus_1.xSensorError;
(* STLV59_A_360_014_SQ401 *)
FbMpbus_2(xEnable := STLV59_360.STLV59_A_360_014_SQ401.xEnable, bPortMpBus := 1, bAddress := 2, tCycleTime := t#500ms, rAirVolume := STLV59_360.STLV59_A_360_014_SQ401.rAirVolume_SP, rMinAirVolume := 0, rMaxAirVolume := 100, xSet := xSet, xRead := xRead, bSensorType := 0, xManualOpen := STLV59_360.STLV59_A_360_014_SQ401.xManualOpen, xManualClose := STLV59_360.STLV59_A_360_014_SQ401.xManualClose);
oStatus_2 := FbMpbus_2.oStatus;
sStatus_2 := FbMpbus_2.sStatus;
STLV59_360.STLV59_A_360_014_SQ401.xReady := FbMpbus_2.xReady;
STLV59_360.STLV59_A_360_014_SQ401.rOutPosition := FbMpbus_2.rOutPosition;
STLV59_360.STLV59_A_360_014_SQ401.rOutAirVolume_perc := FbMpbus_2.rOutAirVolume_perc;
STLV59_360.STLV59_A_360_014_SQ401.rOutAirVolume_m3h := FbMpbus_2.rOutAirVolume_m3_h;
STLV59_360.STLV59_A_360_014_SQ401.wSensorValue := FbMpbus_2.wSensorValue;
STLV59_360.STLV59_A_360_014_SQ401.rVmin := FbMpbus_2.rVmin;
STLV59_360.STLV59_A_360_014_SQ401.rVmax := FbMpbus_2.rVmax;
STLV59_360.STLV59_A_360_014_SQ401.xControlRangeIncreased := FbMpbus_2.xControlRangeIncreased;
STLV59_360.STLV59_A_360_014_SQ401.xMecanicalOverload := FbMpbus_2.xMecanicalOverload;
STLV59_360.STLV59_A_360_014_SQ401.xActuatorHunting := FbMpbus_2.xActuatorHunting;
STLV59_360.STLV59_A_360_014_SQ401.xSensorError := FbMpbus_2.xSensorError;
(* STLV59_A_360_014_SQ501 *)
FbMpbus_3(xEnable := STLV59_360.STLV59_A_360_014_SQ501.xEnable, bPortMpBus := 1, bAddress := 3, tCycleTime := t#500ms, rAirVolume := STLV59_360.STLV59_A_360_014_SQ501.rAirVolume_SP, rMinAirVolume := 0, rMaxAirVolume := 100, xSet := xSet, xRead := xRead, bSensorType := 0, xManualOpen := STLV59_360.STLV59_A_360_014_SQ501.xManualOpen, xManualClose := STLV59_360.STLV59_A_360_014_SQ501.xManualClose);
oStatus_3 := FbMpbus_3.oStatus;
sStatus_3 := FbMpbus_3.sStatus;
STLV59_360.STLV59_A_360_014_SQ501.xReady := FbMpbus_3.xReady;
STLV59_360.STLV59_A_360_014_SQ501.rOutPosition := FbMpbus_3.rOutPosition;
STLV59_360.STLV59_A_360_014_SQ501.rOutAirVolume_perc := FbMpbus_3.rOutAirVolume_perc;
STLV59_360.STLV59_A_360_014_SQ501.rOutAirVolume_m3h := FbMpbus_3.rOutAirVolume_m3_h;
STLV59_360.STLV59_A_360_014_SQ501.wSensorValue := FbMpbus_3.wSensorValue;
STLV59_360.STLV59_A_360_014_SQ501.rVmin := FbMpbus_3.rVmin;
STLV59_360.STLV59_A_360_014_SQ501.rVmax := FbMpbus_3.rVmax;
STLV59_360.STLV59_A_360_014_SQ501.xControlRangeIncreased := FbMpbus_3.xControlRangeIncreased;
STLV59_360.STLV59_A_360_014_SQ501.xMecanicalOverload := FbMpbus_3.xMecanicalOverload;
STLV59_360.STLV59_A_360_014_SQ501.xActuatorHunting := FbMpbus_3.xActuatorHunting;
STLV59_360.STLV59_A_360_014_SQ501.xSensorError := FbMpbus_3.xSensorError;
(* STLV59_A_360_103_SQ401 *)
FbMpbus_4(xEnable := STLV59_360.STLV59_A_360_103_SQ401.xEnable, bPortMpBus := 1, bAddress := 4, tCycleTime := t#500ms, rAirVolume := STLV59_360.STLV59_A_360_103_SQ401.rAirVolume_SP, rMinAirVolume := 0, rMaxAirVolume := 100, xSet := xSet, xRead := xRead, bSensorType := 0, xManualOpen := STLV59_360.STLV59_A_360_103_SQ401.xManualOpen, xManualClose := STLV59_360.STLV59_A_360_103_SQ401.xManualClose);
oStatus_4 := FbMpbus_4.oStatus;
sStatus_4 := FbMpbus_4.sStatus;
STLV59_360.STLV59_A_360_103_SQ401.xReady := FbMpbus_4.xReady;
STLV59_360.STLV59_A_360_103_SQ401.rOutPosition := FbMpbus_4.rOutPosition;
STLV59_360.STLV59_A_360_103_SQ401.rOutAirVolume_perc := FbMpbus_4.rOutAirVolume_perc;
STLV59_360.STLV59_A_360_103_SQ401.rOutAirVolume_m3h := FbMpbus_4.rOutAirVolume_m3_h;
STLV59_360.STLV59_A_360_103_SQ401.wSensorValue := FbMpbus_4.wSensorValue;
STLV59_360.STLV59_A_360_103_SQ401.rVmin := FbMpbus_4.rVmin;
STLV59_360.STLV59_A_360_103_SQ401.rVmax := FbMpbus_4.rVmax;
STLV59_360.STLV59_A_360_103_SQ401.xControlRangeIncreased := FbMpbus_4.xControlRangeIncreased;
STLV59_360.STLV59_A_360_103_SQ401.xMecanicalOverload := FbMpbus_4.xMecanicalOverload;
STLV59_360.STLV59_A_360_103_SQ401.xActuatorHunting := FbMpbus_4.xActuatorHunting;
STLV59_360.STLV59_A_360_103_SQ401.xSensorError := FbMpbus_4.xSensorError;
(* STLV59_A_360_103_SQ402 *)
FbMpbus_5(xEnable := STLV59_360.STLV59_A_360_103_SQ402.xEnable, bPortMpBus := 1, bAddress := 5, tCycleTime := t#500ms, rAirVolume := STLV59_360.STLV59_A_360_103_SQ402.rAirVolume_SP, rMinAirVolume := 0, rMaxAirVolume := 100, xSet := xSet, xRead := xRead, bSensorType := 0, xManualOpen := STLV59_360.STLV59_A_360_103_SQ402.xManualOpen, xManualClose := STLV59_360.STLV59_A_360_103_SQ402.xManualClose);
oStatus_5 := FbMpbus_5.oStatus;
sStatus_5 := FbMpbus_5.sStatus;
STLV59_360.STLV59_A_360_103_SQ402.xReady := FbMpbus_5.xReady;
STLV59_360.STLV59_A_360_103_SQ402.rOutPosition := FbMpbus_5.rOutPosition;
STLV59_360.STLV59_A_360_103_SQ402.rOutAirVolume_perc := FbMpbus_5.rOutAirVolume_perc;
STLV59_360.STLV59_A_360_103_SQ402.rOutAirVolume_m3h := FbMpbus_5.rOutAirVolume_m3_h;
STLV59_360.STLV59_A_360_103_SQ402.wSensorValue := FbMpbus_5.wSensorValue;
STLV59_360.STLV59_A_360_103_SQ402.rVmin := FbMpbus_5.rVmin;
STLV59_360.STLV59_A_360_103_SQ402.rVmax := FbMpbus_5.rVmax;
STLV59_360.STLV59_A_360_103_SQ402.xControlRangeIncreased := FbMpbus_5.xControlRangeIncreased;
STLV59_360.STLV59_A_360_103_SQ402.xMecanicalOverload := FbMpbus_5.xMecanicalOverload;
STLV59_360.STLV59_A_360_103_SQ402.xActuatorHunting := FbMpbus_5.xActuatorHunting;
STLV59_360.STLV59_A_360_103_SQ402.xSensorError := FbMpbus_5.xSensorError;
(* STLV59_A_360_103_SQ501 *)
FbMpbus_6(xEnable := STLV59_360.STLV59_A_360_103_SQ501.xEnable, bPortMpBus := 1, bAddress := 6, tCycleTime := t#500ms, rAirVolume := STLV59_360.STLV59_A_360_103_SQ501.rAirVolume_SP, rMinAirVolume := 0, rMaxAirVolume := 100, xSet := xSet, xRead := xRead, bSensorType := 0, xManualOpen := STLV59_360.STLV59_A_360_103_SQ501.xManualOpen, xManualClose := STLV59_360.STLV59_A_360_103_SQ501.xManualClose);
oStatus_6 := FbMpbus_6.oStatus;
sStatus_6 := FbMpbus_6.sStatus;
STLV59_360.STLV59_A_360_103_SQ501.xReady := FbMpbus_6.xReady;
STLV59_360.STLV59_A_360_103_SQ501.rOutPosition := FbMpbus_6.rOutPosition;
STLV59_360.STLV59_A_360_103_SQ501.rOutAirVolume_perc := FbMpbus_6.rOutAirVolume_perc;
STLV59_360.STLV59_A_360_103_SQ501.rOutAirVolume_m3h := FbMpbus_6.rOutAirVolume_m3_h;
STLV59_360.STLV59_A_360_103_SQ501.wSensorValue := FbMpbus_6.wSensorValue;
STLV59_360.STLV59_A_360_103_SQ501.rVmin := FbMpbus_6.rVmin;
STLV59_360.STLV59_A_360_103_SQ501.rVmax := FbMpbus_6.rVmax;
STLV59_360.STLV59_A_360_103_SQ501.xControlRangeIncreased := FbMpbus_6.xControlRangeIncreased;
STLV59_360.STLV59_A_360_103_SQ501.xMecanicalOverload := FbMpbus_6.xMecanicalOverload;
STLV59_360.STLV59_A_360_103_SQ501.xActuatorHunting := FbMpbus_6.xActuatorHunting;
STLV59_360.STLV59_A_360_103_SQ501.xSensorError := FbMpbus_6.xSensorError;
(* STLV59_A_360_103_SQ502 *)
FbMpbus_7(xEnable := STLV59_360.STLV59_A_360_103_SQ502.xEnable, bPortMpBus := 1, bAddress := 7, tCycleTime := t#500ms, rAirVolume := STLV59_360.STLV59_A_360_103_SQ502.rAirVolume_SP, rMinAirVolume := 0, rMaxAirVolume := 100, xSet := xSet, xRead := xRead, bSensorType := 0, xManualOpen := STLV59_360.STLV59_A_360_103_SQ502.xManualOpen, xManualClose := STLV59_360.STLV59_A_360_103_SQ502.xManualClose);
oStatus_7 := FbMpbus_7.oStatus;
sStatus_7 := FbMpbus_7.sStatus;
STLV59_360.STLV59_A_360_103_SQ502.xReady := FbMpbus_7.xReady;
STLV59_360.STLV59_A_360_103_SQ502.rOutPosition := FbMpbus_7.rOutPosition;
STLV59_360.STLV59_A_360_103_SQ502.rOutAirVolume_perc := FbMpbus_7.rOutAirVolume_perc;
STLV59_360.STLV59_A_360_103_SQ502.rOutAirVolume_m3h := FbMpbus_7.rOutAirVolume_m3_h;
STLV59_360.STLV59_A_360_103_SQ502.wSensorValue := FbMpbus_7.wSensorValue;
STLV59_360.STLV59_A_360_103_SQ502.rVmin := FbMpbus_7.rVmin;
STLV59_360.STLV59_A_360_103_SQ502.rVmax := FbMpbus_7.rVmax;
STLV59_360.STLV59_A_360_103_SQ502.xControlRangeIncreased := FbMpbus_7.xControlRangeIncreased;
STLV59_360.STLV59_A_360_103_SQ502.xMecanicalOverload := FbMpbus_7.xMecanicalOverload;
STLV59_360.STLV59_A_360_103_SQ502.xActuatorHunting := FbMpbus_7.xActuatorHunting;
STLV59_360.STLV59_A_360_103_SQ502.xSensorError := FbMpbus_7.xSensorError;
END_PROGRAM

PROGRAM PRG_360_MP2
  VAR
    xSet : BOOL;  (* Felles *)
    xRead : BOOL;
    FbMpbusMaster_2 : FbMpbusMaster;  (* Master *)
    oStatus_M2 : WagoSysErrorBase.FbResult;
    sStatus_M2 : STRING;
    FbMpbus_1 : FbMpBusVav;  (* Linje 2. Adresse 1. VAV STLV59_A_360_002_SQ402 *)
    oStatus_1 : WagoSysErrorBase.FbResult;
    sStatus_1 : STRING;
    FbMpbus_2 : FbMpBusVav;  (* Linje 2. Adresse 2. VAV STLV59_A_360_002_SQ501 *)
    oStatus_2 : WagoSysErrorBase.FbResult;
    sStatus_2 : STRING;
    FbMpbus_3 : FbMpBusVav;  (* Linje 2. Adresse 3. VAV STLV59_A_360_002_SQ502 *)
    oStatus_3 : WagoSysErrorBase.FbResult;
    sStatus_3 : STRING;
    FbMpbus_4 : FbMpBusVav;  (* Linje 2. Adresse 4. VAV STLV59_A_360_006_SQ401 *)
    oStatus_4 : WagoSysErrorBase.FbResult;
    sStatus_4 : STRING;
    FbMpbus_5 : FbMpBusVav;  (* Linje 2. Adresse 5. VAV STLV59_A_360_008_SQ501 *)
    oStatus_5 : WagoSysErrorBase.FbResult;
    sStatus_5 : STRING;
    FbMpbus_6 : FbMpBusVav;  (* Linje 2. Adresse 6. VAV STLV59_A_360_011_SQ401 *)
    oStatus_6 : WagoSysErrorBase.FbResult;
    sStatus_6 : STRING;
    FbMpbus_7 : FbMpBusVav;  (* Linje 2. Adresse 7. VAV STLV59_A_360_011_SQ501 *)
    oStatus_7 : WagoSysErrorBase.FbResult;
    sStatus_7 : STRING;
    FbMpbus_8 : FbMpBusVav;  (* Linje 2. Adresse 8. VAV STLV59_A_360_T1U_SQ401 *)
    oStatus_8 : WagoSysErrorBase.FbResult;
    sStatus_8 : STRING;
  END_VAR

(* CFC diagram, written out as Structured Text *)
FbMpbusMaster_2(I_Port := IoConfig_Globals.MP_Bus_Master_1, bPortMpBus := 2);
oStatus_M2 := FbMpbusMaster_2.oStatus;
sStatus_M2 := FbMpbusMaster_2.sStatus;
(* STLV59_A_360_002_SQ402 *)
FbMpbus_1(xEnable := STLV59_360.STLV59_A_360_002_SQ402.xEnable, bPortMpBus := 2, bAddress := 1, tCycleTime := t#500ms, rAirVolume := STLV59_360.STLV59_A_360_002_SQ402.rAirVolume_SP, rMinAirVolume := 0, rMaxAirVolume := 100, xSet := xSet, xRead := xRead, bSensorType := 0, xManualOpen := STLV59_360.STLV59_A_360_002_SQ402.xManualOpen, xManualClose := STLV59_360.STLV59_A_360_002_SQ402.xManualClose);
oStatus_1 := FbMpbus_1.oStatus;
sStatus_1 := FbMpbus_1.sStatus;
STLV59_360.STLV59_A_360_002_SQ402.xReady := FbMpbus_1.xReady;
STLV59_360.STLV59_A_360_002_SQ402.rOutPosition := FbMpbus_1.rOutPosition;
STLV59_360.STLV59_A_360_002_SQ402.rOutAirVolume_perc := FbMpbus_1.rOutAirVolume_perc;
STLV59_360.STLV59_A_360_002_SQ402.rOutAirVolume_m3h := FbMpbus_1.rOutAirVolume_m3_h;
STLV59_360.STLV59_A_360_002_SQ402.wSensorValue := FbMpbus_1.wSensorValue;
STLV59_360.STLV59_A_360_002_SQ402.rVmin := FbMpbus_1.rVmin;
STLV59_360.STLV59_A_360_002_SQ402.rVmax := FbMpbus_1.rVmax;
STLV59_360.STLV59_A_360_002_SQ402.xControlRangeIncreased := FbMpbus_1.xControlRangeIncreased;
STLV59_360.STLV59_A_360_002_SQ402.xMecanicalOverload := FbMpbus_1.xMecanicalOverload;
STLV59_360.STLV59_A_360_002_SQ402.xActuatorHunting := FbMpbus_1.xActuatorHunting;
STLV59_360.STLV59_A_360_002_SQ402.xSensorError := FbMpbus_1.xSensorError;
(* STLV59_A_360_002_SQ501 *)
FbMpbus_2(xEnable := STLV59_360.STLV59_A_360_002_SQ501.xEnable, bPortMpBus := 2, bAddress := 2, tCycleTime := t#500ms, rAirVolume := STLV59_360.STLV59_A_360_002_SQ501.rAirVolume_SP, rMinAirVolume := 0, rMaxAirVolume := 100, xSet := xSet, xRead := xRead, bSensorType := 0, xManualOpen := STLV59_360.STLV59_A_360_002_SQ501.xManualOpen, xManualClose := STLV59_360.STLV59_A_360_002_SQ501.xManualClose);
oStatus_2 := FbMpbus_2.oStatus;
sStatus_2 := FbMpbus_2.sStatus;
STLV59_360.STLV59_A_360_002_SQ501.xReady := FbMpbus_2.xReady;
STLV59_360.STLV59_A_360_002_SQ501.rOutPosition := FbMpbus_2.rOutPosition;
STLV59_360.STLV59_A_360_002_SQ501.rOutAirVolume_perc := FbMpbus_2.rOutAirVolume_perc;
STLV59_360.STLV59_A_360_002_SQ501.rOutAirVolume_m3h := FbMpbus_2.rOutAirVolume_m3_h;
STLV59_360.STLV59_A_360_002_SQ501.wSensorValue := FbMpbus_2.wSensorValue;
STLV59_360.STLV59_A_360_002_SQ501.rVmin := FbMpbus_2.rVmin;
STLV59_360.STLV59_A_360_002_SQ501.rVmax := FbMpbus_2.rVmax;
STLV59_360.STLV59_A_360_002_SQ501.xControlRangeIncreased := FbMpbus_2.xControlRangeIncreased;
STLV59_360.STLV59_A_360_002_SQ501.xMecanicalOverload := FbMpbus_2.xMecanicalOverload;
STLV59_360.STLV59_A_360_002_SQ501.xActuatorHunting := FbMpbus_2.xActuatorHunting;
STLV59_360.STLV59_A_360_002_SQ501.xSensorError := FbMpbus_2.xSensorError;
(* STLV59_A_360_002_SQ502 *)
FbMpbus_3(xEnable := STLV59_360.STLV59_A_360_002_SQ502.xEnable, bPortMpBus := 2, bAddress := 3, tCycleTime := t#500ms, rAirVolume := STLV59_360.STLV59_A_360_002_SQ502.rAirVolume_SP, rMinAirVolume := 0, rMaxAirVolume := 100, xSet := xSet, xRead := xRead, bSensorType := 0, xManualOpen := STLV59_360.STLV59_A_360_002_SQ502.xManualOpen, xManualClose := STLV59_360.STLV59_A_360_002_SQ502.xManualClose);
oStatus_3 := FbMpbus_3.oStatus;
sStatus_3 := FbMpbus_3.sStatus;
STLV59_360.STLV59_A_360_002_SQ502.xReady := FbMpbus_3.xReady;
STLV59_360.STLV59_A_360_002_SQ502.rOutPosition := FbMpbus_3.rOutPosition;
STLV59_360.STLV59_A_360_002_SQ502.rOutAirVolume_perc := FbMpbus_3.rOutAirVolume_perc;
STLV59_360.STLV59_A_360_002_SQ502.rOutAirVolume_m3h := FbMpbus_3.rOutAirVolume_m3_h;
STLV59_360.STLV59_A_360_002_SQ502.wSensorValue := FbMpbus_3.wSensorValue;
STLV59_360.STLV59_A_360_002_SQ502.rVmin := FbMpbus_3.rVmin;
STLV59_360.STLV59_A_360_002_SQ502.rVmax := FbMpbus_3.rVmax;
STLV59_360.STLV59_A_360_002_SQ502.xControlRangeIncreased := FbMpbus_3.xControlRangeIncreased;
STLV59_360.STLV59_A_360_002_SQ502.xMecanicalOverload := FbMpbus_3.xMecanicalOverload;
STLV59_360.STLV59_A_360_002_SQ502.xActuatorHunting := FbMpbus_3.xActuatorHunting;
STLV59_360.STLV59_A_360_002_SQ502.xSensorError := FbMpbus_3.xSensorError;
(* STLV59_A_360_006_SQ401 *)
FbMpbus_4(xEnable := STLV59_360.STLV59_A_360_006_SQ401.xEnable, bPortMpBus := 2, bAddress := 4, tCycleTime := t#500ms, rAirVolume := STLV59_360.STLV59_A_360_006_SQ401.rAirVolume_SP, rMinAirVolume := 0, rMaxAirVolume := 100, xSet := xSet, xRead := xRead, bSensorType := 0, xManualOpen := STLV59_360.STLV59_A_360_006_SQ401.xManualOpen, xManualClose := STLV59_360.STLV59_A_360_006_SQ401.xManualClose);
oStatus_4 := FbMpbus_4.oStatus;
sStatus_4 := FbMpbus_4.sStatus;
STLV59_360.STLV59_A_360_006_SQ401.xReady := FbMpbus_4.xReady;
STLV59_360.STLV59_A_360_006_SQ401.rOutPosition := FbMpbus_4.rOutPosition;
STLV59_360.STLV59_A_360_006_SQ401.rOutAirVolume_perc := FbMpbus_4.rOutAirVolume_perc;
STLV59_360.STLV59_A_360_006_SQ401.rOutAirVolume_m3h := FbMpbus_4.rOutAirVolume_m3_h;
STLV59_360.STLV59_A_360_006_SQ401.wSensorValue := FbMpbus_4.wSensorValue;
STLV59_360.STLV59_A_360_006_SQ401.rVmin := FbMpbus_4.rVmin;
STLV59_360.STLV59_A_360_006_SQ401.rVmax := FbMpbus_4.rVmax;
STLV59_360.STLV59_A_360_006_SQ401.xControlRangeIncreased := FbMpbus_4.xControlRangeIncreased;
STLV59_360.STLV59_A_360_006_SQ401.xMecanicalOverload := FbMpbus_4.xMecanicalOverload;
STLV59_360.STLV59_A_360_006_SQ401.xActuatorHunting := FbMpbus_4.xActuatorHunting;
STLV59_360.STLV59_A_360_006_SQ401.xSensorError := FbMpbus_4.xSensorError;
(* STLV59_A_360_008_SQ501 *)
FbMpbus_5(xEnable := STLV59_360.STLV59_A_360_008_SQ501.xEnable, bPortMpBus := 2, bAddress := 5, tCycleTime := t#500ms, rAirVolume := STLV59_360.STLV59_A_360_008_SQ501.rAirVolume_SP, rMinAirVolume := 0, rMaxAirVolume := 100, xSet := xSet, xRead := xRead, bSensorType := 0, xManualOpen := STLV59_360.STLV59_A_360_008_SQ501.xManualOpen, xManualClose := STLV59_360.STLV59_A_360_008_SQ501.xManualClose);
oStatus_5 := FbMpbus_5.oStatus;
sStatus_5 := FbMpbus_5.sStatus;
STLV59_360.STLV59_A_360_008_SQ501.xReady := FbMpbus_5.xReady;
STLV59_360.STLV59_A_360_008_SQ501.rOutPosition := FbMpbus_5.rOutPosition;
STLV59_360.STLV59_A_360_008_SQ501.rOutAirVolume_perc := FbMpbus_5.rOutAirVolume_perc;
STLV59_360.STLV59_A_360_008_SQ501.rOutAirVolume_m3h := FbMpbus_5.rOutAirVolume_m3_h;
STLV59_360.STLV59_A_360_008_SQ501.wSensorValue := FbMpbus_5.wSensorValue;
STLV59_360.STLV59_A_360_008_SQ501.rVmin := FbMpbus_5.rVmin;
STLV59_360.STLV59_A_360_008_SQ501.rVmax := FbMpbus_5.rVmax;
STLV59_360.STLV59_A_360_008_SQ501.xControlRangeIncreased := FbMpbus_5.xControlRangeIncreased;
STLV59_360.STLV59_A_360_008_SQ501.xMecanicalOverload := FbMpbus_5.xMecanicalOverload;
STLV59_360.STLV59_A_360_008_SQ501.xActuatorHunting := FbMpbus_5.xActuatorHunting;
STLV59_360.STLV59_A_360_008_SQ501.xSensorError := FbMpbus_5.xSensorError;
(* STLV59_A_360_011_SQ401 *)
FbMpbus_6(xEnable := STLV59_360.STLV59_A_360_011_SQ401.xEnable, bPortMpBus := 2, bAddress := 6, tCycleTime := t#500ms, rAirVolume := STLV59_360.STLV59_A_360_011_SQ401.rAirVolume_SP, rMinAirVolume := 0, rMaxAirVolume := 100, xSet := xSet, xRead := xRead, bSensorType := 0, xManualOpen := STLV59_360.STLV59_A_360_011_SQ401.xManualOpen, xManualClose := STLV59_360.STLV59_A_360_011_SQ401.xManualClose);
oStatus_6 := FbMpbus_6.oStatus;
sStatus_6 := FbMpbus_6.sStatus;
STLV59_360.STLV59_A_360_011_SQ401.xReady := FbMpbus_6.xReady;
STLV59_360.STLV59_A_360_011_SQ401.rOutPosition := FbMpbus_6.rOutPosition;
STLV59_360.STLV59_A_360_011_SQ401.rOutAirVolume_perc := FbMpbus_6.rOutAirVolume_perc;
STLV59_360.STLV59_A_360_011_SQ401.rOutAirVolume_m3h := FbMpbus_6.rOutAirVolume_m3_h;
STLV59_360.STLV59_A_360_011_SQ401.wSensorValue := FbMpbus_6.wSensorValue;
STLV59_360.STLV59_A_360_011_SQ401.rVmin := FbMpbus_6.rVmin;
STLV59_360.STLV59_A_360_011_SQ401.rVmax := FbMpbus_6.rVmax;
STLV59_360.STLV59_A_360_011_SQ401.xControlRangeIncreased := FbMpbus_6.xControlRangeIncreased;
STLV59_360.STLV59_A_360_011_SQ401.xMecanicalOverload := FbMpbus_6.xMecanicalOverload;
STLV59_360.STLV59_A_360_011_SQ401.xActuatorHunting := FbMpbus_6.xActuatorHunting;
STLV59_360.STLV59_A_360_011_SQ401.xSensorError := FbMpbus_6.xSensorError;
(* STLV59_A_360_011_SQ501 *)
FbMpbus_7(xEnable := STLV59_360.STLV59_A_360_011_SQ501.xEnable, bPortMpBus := 2, bAddress := 7, tCycleTime := t#500ms, rAirVolume := STLV59_360.STLV59_A_360_011_SQ501.rAirVolume_SP, rMinAirVolume := 0, rMaxAirVolume := 100, xSet := xSet, xRead := xRead, bSensorType := 0, xManualOpen := STLV59_360.STLV59_A_360_011_SQ501.xManualOpen, xManualClose := STLV59_360.STLV59_A_360_011_SQ501.xManualClose);
oStatus_7 := FbMpbus_7.oStatus;
sStatus_7 := FbMpbus_7.sStatus;
STLV59_360.STLV59_A_360_011_SQ501.xReady := FbMpbus_7.xReady;
STLV59_360.STLV59_A_360_011_SQ501.rOutPosition := FbMpbus_7.rOutPosition;
STLV59_360.STLV59_A_360_011_SQ501.rOutAirVolume_perc := FbMpbus_7.rOutAirVolume_perc;
STLV59_360.STLV59_A_360_011_SQ501.rOutAirVolume_m3h := FbMpbus_7.rOutAirVolume_m3_h;
STLV59_360.STLV59_A_360_011_SQ501.wSensorValue := FbMpbus_7.wSensorValue;
STLV59_360.STLV59_A_360_011_SQ501.rVmin := FbMpbus_7.rVmin;
STLV59_360.STLV59_A_360_011_SQ501.rVmax := FbMpbus_7.rVmax;
STLV59_360.STLV59_A_360_011_SQ501.xControlRangeIncreased := FbMpbus_7.xControlRangeIncreased;
STLV59_360.STLV59_A_360_011_SQ501.xMecanicalOverload := FbMpbus_7.xMecanicalOverload;
STLV59_360.STLV59_A_360_011_SQ501.xActuatorHunting := FbMpbus_7.xActuatorHunting;
STLV59_360.STLV59_A_360_011_SQ501.xSensorError := FbMpbus_7.xSensorError;
(* STLV59_A_360_T1U_SQ401 *)
FbMpbus_8(xEnable := STLV59_360.STLV59_A_360_T1U_SQ401.xEnable, bPortMpBus := 2, bAddress := 8, tCycleTime := t#500ms, rAirVolume := STLV59_360.STLV59_A_360_T1U_SQ401.rAirVolume_SP, rMinAirVolume := 0, rMaxAirVolume := 100, xSet := xSet, xRead := xRead, bSensorType := 0, xManualOpen := STLV59_360.STLV59_A_360_T1U_SQ401.xManualOpen, xManualClose := STLV59_360.STLV59_A_360_T1U_SQ401.xManualClose);
oStatus_8 := FbMpbus_8.oStatus;
sStatus_8 := FbMpbus_8.sStatus;
STLV59_360.STLV59_A_360_T1U_SQ401.xReady := FbMpbus_8.xReady;
STLV59_360.STLV59_A_360_T1U_SQ401.rOutPosition := FbMpbus_8.rOutPosition;
STLV59_360.STLV59_A_360_T1U_SQ401.rOutAirVolume_perc := FbMpbus_8.rOutAirVolume_perc;
STLV59_360.STLV59_A_360_T1U_SQ401.rOutAirVolume_m3h := FbMpbus_8.rOutAirVolume_m3_h;
STLV59_360.STLV59_A_360_T1U_SQ401.wSensorValue := FbMpbus_8.wSensorValue;
STLV59_360.STLV59_A_360_T1U_SQ401.rVmin := FbMpbus_8.rVmin;
STLV59_360.STLV59_A_360_T1U_SQ401.rVmax := FbMpbus_8.rVmax;
STLV59_360.STLV59_A_360_T1U_SQ401.xControlRangeIncreased := FbMpbus_8.xControlRangeIncreased;
STLV59_360.STLV59_A_360_T1U_SQ401.xMecanicalOverload := FbMpbus_8.xMecanicalOverload;
STLV59_360.STLV59_A_360_T1U_SQ401.xActuatorHunting := FbMpbus_8.xActuatorHunting;
STLV59_360.STLV59_A_360_T1U_SQ401.xSensorError := FbMpbus_8.xSensorError;
END_PROGRAM

PROGRAM PRG_360_MP3
  VAR
    xSet : BOOL;  (* Felles *)
    xRead : BOOL;
    FbMpbusMaster_3 : FbMpbusMaster;  (* Master *)
    oStatus_M3 : WagoSysErrorBase.FbResult;
    sStatus_M3 : STRING;
    FbMpbus_1 : FbMpBusVav;  (* Linje 3. Adresse 1. VAV STLV59_A_360_001_SQ401 *)
    oStatus_1 : WagoSysErrorBase.FbResult;
    sStatus_1 : STRING;
    FbMpbus_2 : FbMpBusVav;  (* Linje 3. Adresse 2. VAV STLV59_A_360_001_SQ501 *)
    oStatus_2 : WagoSysErrorBase.FbResult;
    sStatus_2 : STRING;
    FbMpbus_3 : FbMpBusVav;  (* Linje 3. Adresse 3. VAV STLV59_A_360_109_SQ401 *)
    oStatus_3 : WagoSysErrorBase.FbResult;
    sStatus_3 : STRING;
    FbMpbus_4 : FbMpBusVav;  (* Linje 3. Adresse 4. VAV STLV59_A_360_110_SQ501 *)
    oStatus_4 : WagoSysErrorBase.FbResult;
    sStatus_4 : STRING;
    FbMpbus_5 : FbMpBusVav;  (* Linje 3. Adresse 5. VAV STLV59_A_360_212_SQ401 *)
    oStatus_5 : WagoSysErrorBase.FbResult;
    sStatus_5 : STRING;
    FbMpbus_6 : FbMpBusVav;  (* Linje 3. Adresse 6. VAV STLV59_A_360_212_SQ501 *)
    oStatus_6 : WagoSysErrorBase.FbResult;
    sStatus_6 : STRING;
    FbMpbus_7 : FbMpBusVav;  (* Linje 3. Adresse 7. VAV STLV59_A_360_213_SQ401 *)
    oStatus_7 : WagoSysErrorBase.FbResult;
    sStatus_7 : STRING;
    FbMpbus_8 : FbMpBusVav;  (* Linje 3. Adresse 8. VAV STLV59_A_360_213_SQ501 *)
    oStatus_8 : WagoSysErrorBase.FbResult;
    sStatus_8 : STRING;
  END_VAR

(* CFC diagram, written out as Structured Text *)
FbMpbusMaster_3(I_Port := IoConfig_Globals.MP_Bus_Master_2, bPortMpBus := 3);
oStatus_M3 := FbMpbusMaster_3.oStatus;
sStatus_M3 := FbMpbusMaster_3.sStatus;
(* STLV59_A_360_001_SQ401 *)
FbMpbus_1(xEnable := STLV59_360.STLV59_A_360_001_SQ401.xEnable, bPortMpBus := 3, bAddress := 1, tCycleTime := t#500ms, rAirVolume := STLV59_360.STLV59_A_360_001_SQ401.rAirVolume_SP, rMinAirVolume := 0, rMaxAirVolume := 100, xSet := xSet, xRead := xRead, bSensorType := 0, xManualOpen := STLV59_360.STLV59_A_360_001_SQ401.xManualOpen, xManualClose := STLV59_360.STLV59_A_360_001_SQ401.xManualClose);
oStatus_1 := FbMpbus_1.oStatus;
sStatus_1 := FbMpbus_1.sStatus;
STLV59_360.STLV59_A_360_001_SQ401.xReady := FbMpbus_1.xReady;
STLV59_360.STLV59_A_360_001_SQ401.rOutPosition := FbMpbus_1.rOutPosition;
STLV59_360.STLV59_A_360_001_SQ401.rOutAirVolume_perc := FbMpbus_1.rOutAirVolume_perc;
STLV59_360.STLV59_A_360_001_SQ401.rOutAirVolume_m3h := FbMpbus_1.rOutAirVolume_m3_h;
STLV59_360.STLV59_A_360_001_SQ401.wSensorValue := FbMpbus_1.wSensorValue;
STLV59_360.STLV59_A_360_001_SQ401.rVmin := FbMpbus_1.rVmin;
STLV59_360.STLV59_A_360_001_SQ401.rVmax := FbMpbus_1.rVmax;
STLV59_360.STLV59_A_360_001_SQ401.xControlRangeIncreased := FbMpbus_1.xControlRangeIncreased;
STLV59_360.STLV59_A_360_001_SQ401.xMecanicalOverload := FbMpbus_1.xMecanicalOverload;
STLV59_360.STLV59_A_360_001_SQ401.xActuatorHunting := FbMpbus_1.xActuatorHunting;
STLV59_360.STLV59_A_360_001_SQ401.xSensorError := FbMpbus_1.xSensorError;
(* STLV59_A_360_001_SQ501 *)
FbMpbus_2(xEnable := STLV59_360.STLV59_A_360_001_SQ501.xEnable, bPortMpBus := 3, bAddress := 2, tCycleTime := t#500ms, rAirVolume := STLV59_360.STLV59_A_360_001_SQ501.rAirVolume_SP, rMinAirVolume := 0, rMaxAirVolume := 100, xSet := xSet, xRead := xRead, bSensorType := 0, xManualOpen := STLV59_360.STLV59_A_360_001_SQ501.xManualOpen, xManualClose := STLV59_360.STLV59_A_360_001_SQ501.xManualClose);
oStatus_2 := FbMpbus_2.oStatus;
sStatus_2 := FbMpbus_2.sStatus;
STLV59_360.STLV59_A_360_001_SQ501.xReady := FbMpbus_2.xReady;
STLV59_360.STLV59_A_360_001_SQ501.rOutPosition := FbMpbus_2.rOutPosition;
STLV59_360.STLV59_A_360_001_SQ501.rOutAirVolume_perc := FbMpbus_2.rOutAirVolume_perc;
STLV59_360.STLV59_A_360_001_SQ501.rOutAirVolume_m3h := FbMpbus_2.rOutAirVolume_m3_h;
STLV59_360.STLV59_A_360_001_SQ501.wSensorValue := FbMpbus_2.wSensorValue;
STLV59_360.STLV59_A_360_001_SQ501.rVmin := FbMpbus_2.rVmin;
STLV59_360.STLV59_A_360_001_SQ501.rVmax := FbMpbus_2.rVmax;
STLV59_360.STLV59_A_360_001_SQ501.xControlRangeIncreased := FbMpbus_2.xControlRangeIncreased;
STLV59_360.STLV59_A_360_001_SQ501.xMecanicalOverload := FbMpbus_2.xMecanicalOverload;
STLV59_360.STLV59_A_360_001_SQ501.xActuatorHunting := FbMpbus_2.xActuatorHunting;
STLV59_360.STLV59_A_360_001_SQ501.xSensorError := FbMpbus_2.xSensorError;
(* STLV59_A_360_109_SQ401 *)
FbMpbus_3(xEnable := STLV59_360.STLV59_A_360_109_SQ401.xEnable, bPortMpBus := 3, bAddress := 3, tCycleTime := t#500ms, rAirVolume := STLV59_360.STLV59_A_360_109_SQ401.rAirVolume_SP, rMinAirVolume := 0, rMaxAirVolume := 100, xSet := xSet, xRead := xRead, bSensorType := 0, xManualOpen := STLV59_360.STLV59_A_360_109_SQ401.xManualOpen, xManualClose := STLV59_360.STLV59_A_360_109_SQ401.xManualClose);
oStatus_3 := FbMpbus_3.oStatus;
sStatus_3 := FbMpbus_3.sStatus;
STLV59_360.STLV59_A_360_109_SQ401.xReady := FbMpbus_3.xReady;
STLV59_360.STLV59_A_360_109_SQ401.rOutPosition := FbMpbus_3.rOutPosition;
STLV59_360.STLV59_A_360_109_SQ401.rOutAirVolume_perc := FbMpbus_3.rOutAirVolume_perc;
STLV59_360.STLV59_A_360_109_SQ401.rOutAirVolume_m3h := FbMpbus_3.rOutAirVolume_m3_h;
STLV59_360.STLV59_A_360_109_SQ401.wSensorValue := FbMpbus_3.wSensorValue;
STLV59_360.STLV59_A_360_109_SQ401.rVmin := FbMpbus_3.rVmin;
STLV59_360.STLV59_A_360_109_SQ401.rVmax := FbMpbus_3.rVmax;
STLV59_360.STLV59_A_360_109_SQ401.xControlRangeIncreased := FbMpbus_3.xControlRangeIncreased;
STLV59_360.STLV59_A_360_109_SQ401.xMecanicalOverload := FbMpbus_3.xMecanicalOverload;
STLV59_360.STLV59_A_360_109_SQ401.xActuatorHunting := FbMpbus_3.xActuatorHunting;
STLV59_360.STLV59_A_360_109_SQ401.xSensorError := FbMpbus_3.xSensorError;
(* STLV59_A_360_110_SQ501 *)
FbMpbus_4(xEnable := STLV59_360.STLV59_A_360_110_SQ501.xEnable, bPortMpBus := 3, bAddress := 4, tCycleTime := t#500ms, rAirVolume := STLV59_360.STLV59_A_360_110_SQ501.rAirVolume_SP, rMinAirVolume := 0, rMaxAirVolume := 100, xSet := xSet, xRead := xRead, bSensorType := 0, xManualOpen := STLV59_360.STLV59_A_360_110_SQ501.xManualOpen, xManualClose := STLV59_360.STLV59_A_360_110_SQ501.xManualClose);
oStatus_4 := FbMpbus_4.oStatus;
sStatus_4 := FbMpbus_4.sStatus;
STLV59_360.STLV59_A_360_110_SQ501.xReady := FbMpbus_4.xReady;
STLV59_360.STLV59_A_360_110_SQ501.rOutPosition := FbMpbus_4.rOutPosition;
STLV59_360.STLV59_A_360_110_SQ501.rOutAirVolume_perc := FbMpbus_4.rOutAirVolume_perc;
STLV59_360.STLV59_A_360_110_SQ501.rOutAirVolume_m3h := FbMpbus_4.rOutAirVolume_m3_h;
STLV59_360.STLV59_A_360_110_SQ501.wSensorValue := FbMpbus_4.wSensorValue;
STLV59_360.STLV59_A_360_110_SQ501.rVmin := FbMpbus_4.rVmin;
STLV59_360.STLV59_A_360_110_SQ501.rVmax := FbMpbus_4.rVmax;
STLV59_360.STLV59_A_360_110_SQ501.xControlRangeIncreased := FbMpbus_4.xControlRangeIncreased;
STLV59_360.STLV59_A_360_110_SQ501.xMecanicalOverload := FbMpbus_4.xMecanicalOverload;
STLV59_360.STLV59_A_360_110_SQ501.xActuatorHunting := FbMpbus_4.xActuatorHunting;
STLV59_360.STLV59_A_360_110_SQ501.xSensorError := FbMpbus_4.xSensorError;
(* STLV59_A_360_212_SQ401 *)
FbMpbus_5(xEnable := STLV59_360.STLV59_A_360_212_SQ401.xEnable, bPortMpBus := 3, bAddress := 5, tCycleTime := t#500ms, rAirVolume := STLV59_360.STLV59_A_360_212_SQ401.rAirVolume_SP, rMinAirVolume := 0, rMaxAirVolume := 100, xSet := xSet, xRead := xRead, bSensorType := 0, xManualOpen := STLV59_360.STLV59_A_360_212_SQ401.xManualOpen, xManualClose := STLV59_360.STLV59_A_360_212_SQ401.xManualClose);
oStatus_5 := FbMpbus_5.oStatus;
sStatus_5 := FbMpbus_5.sStatus;
STLV59_360.STLV59_A_360_212_SQ401.xReady := FbMpbus_5.xReady;
STLV59_360.STLV59_A_360_212_SQ401.rOutPosition := FbMpbus_5.rOutPosition;
STLV59_360.STLV59_A_360_212_SQ401.rOutAirVolume_perc := FbMpbus_5.rOutAirVolume_perc;
STLV59_360.STLV59_A_360_212_SQ401.rOutAirVolume_m3h := FbMpbus_5.rOutAirVolume_m3_h;
STLV59_360.STLV59_A_360_212_SQ401.wSensorValue := FbMpbus_5.wSensorValue;
STLV59_360.STLV59_A_360_212_SQ401.rVmin := FbMpbus_5.rVmin;
STLV59_360.STLV59_A_360_212_SQ401.rVmax := FbMpbus_5.rVmax;
STLV59_360.STLV59_A_360_212_SQ401.xControlRangeIncreased := FbMpbus_5.xControlRangeIncreased;
STLV59_360.STLV59_A_360_212_SQ401.xMecanicalOverload := FbMpbus_5.xMecanicalOverload;
STLV59_360.STLV59_A_360_212_SQ401.xActuatorHunting := FbMpbus_5.xActuatorHunting;
STLV59_360.STLV59_A_360_212_SQ401.xSensorError := FbMpbus_5.xSensorError;
(* STLV59_A_360_212_SQ501 *)
FbMpbus_6(xEnable := STLV59_360.STLV59_A_360_212_SQ501.xEnable, bPortMpBus := 3, bAddress := 6, tCycleTime := t#500ms, rAirVolume := STLV59_360.STLV59_A_360_212_SQ501.rAirVolume_SP, rMinAirVolume := 0, rMaxAirVolume := 100, xSet := xSet, xRead := xRead, bSensorType := 0, xManualOpen := STLV59_360.STLV59_A_360_212_SQ501.xManualOpen, xManualClose := STLV59_360.STLV59_A_360_212_SQ501.xManualClose);
oStatus_6 := FbMpbus_6.oStatus;
sStatus_6 := FbMpbus_6.sStatus;
STLV59_360.STLV59_A_360_212_SQ501.xReady := FbMpbus_6.xReady;
STLV59_360.STLV59_A_360_212_SQ501.rOutPosition := FbMpbus_6.rOutPosition;
STLV59_360.STLV59_A_360_212_SQ501.rOutAirVolume_perc := FbMpbus_6.rOutAirVolume_perc;
STLV59_360.STLV59_A_360_212_SQ501.rOutAirVolume_m3h := FbMpbus_6.rOutAirVolume_m3_h;
STLV59_360.STLV59_A_360_212_SQ501.wSensorValue := FbMpbus_6.wSensorValue;
STLV59_360.STLV59_A_360_212_SQ501.rVmin := FbMpbus_6.rVmin;
STLV59_360.STLV59_A_360_212_SQ501.rVmax := FbMpbus_6.rVmax;
STLV59_360.STLV59_A_360_212_SQ501.xControlRangeIncreased := FbMpbus_6.xControlRangeIncreased;
STLV59_360.STLV59_A_360_212_SQ501.xMecanicalOverload := FbMpbus_6.xMecanicalOverload;
STLV59_360.STLV59_A_360_212_SQ501.xActuatorHunting := FbMpbus_6.xActuatorHunting;
STLV59_360.STLV59_A_360_212_SQ501.xSensorError := FbMpbus_6.xSensorError;
(* STLV59_A_360_213_SQ401 *)
FbMpbus_7(xEnable := STLV59_360.STLV59_A_360_213_SQ401.xEnable, bPortMpBus := 3, bAddress := 7, tCycleTime := t#500ms, rAirVolume := STLV59_360.STLV59_A_360_213_SQ401.rAirVolume_SP, rMinAirVolume := 0, rMaxAirVolume := 100, xSet := xSet, xRead := xRead, bSensorType := 0, xManualOpen := STLV59_360.STLV59_A_360_213_SQ401.xManualOpen, xManualClose := STLV59_360.STLV59_A_360_213_SQ401.xManualClose);
oStatus_7 := FbMpbus_7.oStatus;
sStatus_7 := FbMpbus_7.sStatus;
STLV59_360.STLV59_A_360_213_SQ401.xReady := FbMpbus_7.xReady;
STLV59_360.STLV59_A_360_213_SQ401.rOutPosition := FbMpbus_7.rOutPosition;
STLV59_360.STLV59_A_360_213_SQ401.rOutAirVolume_perc := FbMpbus_7.rOutAirVolume_perc;
STLV59_360.STLV59_A_360_213_SQ401.rOutAirVolume_m3h := FbMpbus_7.rOutAirVolume_m3_h;
STLV59_360.STLV59_A_360_213_SQ401.wSensorValue := FbMpbus_7.wSensorValue;
STLV59_360.STLV59_A_360_213_SQ401.rVmin := FbMpbus_7.rVmin;
STLV59_360.STLV59_A_360_213_SQ401.rVmax := FbMpbus_7.rVmax;
STLV59_360.STLV59_A_360_213_SQ401.xControlRangeIncreased := FbMpbus_7.xControlRangeIncreased;
STLV59_360.STLV59_A_360_213_SQ401.xMecanicalOverload := FbMpbus_7.xMecanicalOverload;
STLV59_360.STLV59_A_360_213_SQ401.xActuatorHunting := FbMpbus_7.xActuatorHunting;
STLV59_360.STLV59_A_360_213_SQ401.xSensorError := FbMpbus_7.xSensorError;
(* STLV59_A_360_213_SQ501 *)
FbMpbus_8(xEnable := STLV59_360.STLV59_A_360_213_SQ501.xEnable, bPortMpBus := 3, bAddress := 8, tCycleTime := t#500ms, rAirVolume := STLV59_360.STLV59_A_360_213_SQ501.rAirVolume_SP, rMinAirVolume := 0, rMaxAirVolume := 100, xSet := xSet, xRead := xRead, bSensorType := 0, xManualOpen := STLV59_360.STLV59_A_360_213_SQ501.xManualOpen, xManualClose := STLV59_360.STLV59_A_360_213_SQ501.xManualClose);
oStatus_8 := FbMpbus_8.oStatus;
sStatus_8 := FbMpbus_8.sStatus;
STLV59_360.STLV59_A_360_213_SQ501.xReady := FbMpbus_8.xReady;
STLV59_360.STLV59_A_360_213_SQ501.rOutPosition := FbMpbus_8.rOutPosition;
STLV59_360.STLV59_A_360_213_SQ501.rOutAirVolume_perc := FbMpbus_8.rOutAirVolume_perc;
STLV59_360.STLV59_A_360_213_SQ501.rOutAirVolume_m3h := FbMpbus_8.rOutAirVolume_m3_h;
STLV59_360.STLV59_A_360_213_SQ501.wSensorValue := FbMpbus_8.wSensorValue;
STLV59_360.STLV59_A_360_213_SQ501.rVmin := FbMpbus_8.rVmin;
STLV59_360.STLV59_A_360_213_SQ501.rVmax := FbMpbus_8.rVmax;
STLV59_360.STLV59_A_360_213_SQ501.xControlRangeIncreased := FbMpbus_8.xControlRangeIncreased;
STLV59_360.STLV59_A_360_213_SQ501.xMecanicalOverload := FbMpbus_8.xMecanicalOverload;
STLV59_360.STLV59_A_360_213_SQ501.xActuatorHunting := FbMpbus_8.xActuatorHunting;
STLV59_360.STLV59_A_360_213_SQ501.xSensorError := FbMpbus_8.xSensorError;
END_PROGRAM

PROGRAM PRG_360_VAV_Max

					//Max spjeld vinkel for tilluftsspjeld
STLV59_360.STLV59_A_360_001_OU001_SQ401_Max:=MAX
(
	SEL(STLV59_360.STLV59_A_360_002_SQ401.xdontoptimize, STLV59_360.STLV59_A_360_002_SQ401.rOutPosition, 0),
	SEL(STLV59_360.STLV59_A_360_014_SQ401.xdontoptimize, STLV59_360.STLV59_A_360_014_SQ401.rOutPosition, 0),
	SEL(STLV59_360.STLV59_A_360_103_SQ401.xdontoptimize, STLV59_360.STLV59_A_360_103_SQ401.rOutPosition, 0),
	SEL(STLV59_360.STLV59_A_360_103_SQ402.xdontoptimize, STLV59_360.STLV59_A_360_103_SQ402.rOutPosition, 0),
	SEL(STLV59_360.STLV59_A_360_002_SQ402.xdontoptimize, STLV59_360.STLV59_A_360_002_SQ402.rOutPosition, 0),
	SEL(STLV59_360.STLV59_A_360_006_SQ401.xdontoptimize, STLV59_360.STLV59_A_360_006_SQ401.rOutPosition, 0),
	SEL(STLV59_360.STLV59_A_360_011_SQ401.xdontoptimize, STLV59_360.STLV59_A_360_011_SQ401.rOutPosition, 0),
	SEL(STLV59_360.STLV59_A_360_T1U_SQ401.xdontoptimize, STLV59_360.STLV59_A_360_T1U_SQ401.rOutPosition, 0),
	SEL(STLV59_360.STLV59_A_360_001_SQ401.xdontoptimize, STLV59_360.STLV59_A_360_001_SQ401.rOutPosition, 0),
	SEL(STLV59_360.STLV59_A_360_212_SQ401.xdontoptimize, STLV59_360.STLV59_A_360_212_SQ401.rOutPosition, 0),
	SEL(STLV59_360.STLV59_A_360_213_SQ401.xdontoptimize, STLV59_360.STLV59_A_360_213_SQ401.rOutPosition, 0)
);

//Max spjeld vinkel for avtrekksspjeld
STLV59_360.STLV59_A_360_001_OU001_SQ501_Max:=MAX
(
	SEL(STLV59_360.STLV59_A_360_014_SQ501.xdontoptimize, STLV59_360.STLV59_A_360_014_SQ501.rOutPosition, 0),
	SEL(STLV59_360.STLV59_A_360_103_SQ501.xdontoptimize, STLV59_360.STLV59_A_360_103_SQ501.rOutPosition, 0),
	SEL(STLV59_360.STLV59_A_360_103_SQ502.xdontoptimize, STLV59_360.STLV59_A_360_103_SQ502.rOutPosition, 0),
	SEL(STLV59_360.STLV59_A_360_002_SQ501.xdontoptimize, STLV59_360.STLV59_A_360_002_SQ501.rOutPosition, 0),
	SEL(STLV59_360.STLV59_A_360_002_SQ502.xdontoptimize, STLV59_360.STLV59_A_360_002_SQ502.rOutPosition, 0),
	SEL(STLV59_360.STLV59_A_360_008_SQ501.xdontoptimize, STLV59_360.STLV59_A_360_008_SQ501.rOutPosition, 0),
	SEL(STLV59_360.STLV59_A_360_011_SQ501.xdontoptimize, STLV59_360.STLV59_A_360_011_SQ501.rOutPosition, 0),
	SEL(STLV59_360.STLV59_A_360_001_SQ501.xdontoptimize, STLV59_360.STLV59_A_360_001_SQ501.rOutPosition, 0),
	SEL(STLV59_360.STLV59_A_360_212_SQ501.xdontoptimize, STLV59_360.STLV59_A_360_212_SQ501.rOutPosition, 0),
	SEL(STLV59_360.STLV59_A_360_213_SQ501.xdontoptimize, STLV59_360.STLV59_A_360_213_SQ501.rOutPosition, 0)
);


				
END_PROGRAM
